// TwinCAT 3 PLC project PlantSimulator
// ProgramVersion: 3.1.4026.10
// libraries:
//   Tc2_Standard, * (Beckhoff Automation GmbH)
//   Tc2_System, * (Beckhoff Automation GmbH)
//   Tc3_Module, * (Beckhoff Automation GmbH)
// project tree:
//   / PlcTask.TcTTO
//   POUs/ MAIN.TcPOU, PlantNo1.TcPOU, PlantNo2.TcPOU
// (motion and I/O tree: see PLC project firstplc)
// real-time tasks:
//   TASK PlcTask: cycle T#1ms, priority 20, ADS port 350
//   TASK PlcTask1: cycle T#1ms, priority 21, ADS port 351
// variable links:
//   FirstPLC/FirstPLC Instance <-> PlantSimulator/PlantSimulator Instance
//     PlcTask Inputs/MAIN.lrActualPosition <-> PlcTask Outputs/MAIN.lrOutput
//     PlcTask Outputs/MAIN.lrControllerOutput <-> PlcTask Inputs/MAIN.lrIn

CONFIGURATION PlantSimulator
    RESOURCE PLC ON TwinCAT3
        TASK PlcTask(INTERVAL := T#1ms, PRIORITY := 21);
        PROGRAM MAIN WITH PlcTask : MAIN;
    END_RESOURCE
END_CONFIGURATION

// ---- POUs/MAIN.TcPOU
PROGRAM MAIN
VAR
	lrIn AT%I* : LREAL := 0;
	nCheckCount : INT := 0;
	
	fbPlantNo1: PlantNo1;
	fbPlantNo2: PlantNo2;
	lrOutput AT%Q* : LREAL := 0.0;
	
	nPlant :INT := 0;
	
	lrTempOutput : LREAL := 0.0;
	
	
END_VAR

CASE nPlant OF
	10:
		fbPlantNo1(lrInput := lrIn,
		lrOutput => lrOutput);
		
	20:
		fbPlantNo2(lrInput := lrIn,
			lrM := 3.5,
			lrC := 10,
		lrOutput => lrOutput);
		
	30:
		fbPlantNo1(lrInput := lrIn,
			lrOutput => lrTempOutput);
		fbPlantNo2(lrInput := lrTempOutput,
			lrM := 3.5,
			lrC := 10,
			lrOutput => lrOutput);
			
END_CASE

END_PROGRAM

// ---- POUs/PlantNo1.TcPOU
FUNCTION_BLOCK PlantNo1
VAR_INPUT
	lrInput : LREAL := 0.0;	
END_VAR

VAR_OUTPUT
	lrOutput : LREAL := 0.0;
END_VAR

VAR
	lrLastInput : LREAL := 0.0;
	lrLastOutput : LREAL := 0.0;
	lrTs : LREAL := 0.001;
	lr2OverTs : lreal := 2/0.001;
END_VAR

lr2OverTs := 2.0 / lrTs;
lrOutput := ((lr2OverTs - 500.0) * lrLastOutput + 500.0 * (lrInput + lrLastInput)) / (lr2OverTs + 500.0);
lrLastOutput := lrOutput;
lrLastInput := lrInput;

END_FUNCTION_BLOCK

// ---- POUs/PlantNo2.TcPOU
FUNCTION_BLOCK PlantNo2
VAR_INPUT
	lrInput : LREAL := 0.0;	
	
	lrM : LREAL := 4.72;
	lrC : LREAL := 2.9657;
	
	
END_VAR

VAR_OUTPUT
	lrOutput : LREAL := 0.0;
END_VAR

VAR
	arAccelerationHistory : ARRAY[0..5] OF LREAL := [0.0, 0.0, 0, 0, 0, 0];
	arVeloHistory : ARRAY[0..5] OF LREAL := [0.0, 0.0, 0, 0, 0, 0];
	arPositionHistory : ARRAY[0..5] OF LREAL := [0.0, 0.0, 0, 0, 0, 0];
	nCounter : INT := 0;

	lrTs : LREAL := 0.001;
END_VAR



FOR nCounter := 0 TO 4 DO
	arPositionHistory [5 - nCounter] := arPositionHistory[ 5 - nCounter -1];
	arVeloHistory [5 - nCounter] := arVeloHistory[ 5 - nCounter -1];
	arAccelerationHistory [5 - nCounter] := arAccelerationHistory[ 5 - nCounter -1];
END_FOR


arAccelerationHistory[0] := lrInput / lrM - lrC * arVeloHistory[0] / lrM;

arVeloHistory[0] := arVeloHistory[0] + 0.5 * lrTs * (arAccelerationHistory[0]+arAccelerationHistory[1]);

arPositionHistory[0] := arPositionHistory[0] + 0.5 * lrTs * (arVeloHistory[0]+arVeloHistory[1]);

lrOutput := arPositionHistory[0];

END_FUNCTION_BLOCK
